FUNCTION_BLOCK SufficientFeedFlow (* CAT Function Block Type *)
  (* Standard: 61499-2 *)
  (* Version 0.0, 9/23/2026, Schneider Electric, template *)
  PACKAGE SE.Nereda;
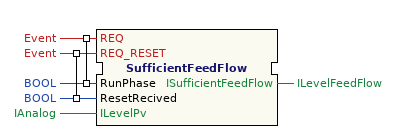
  EVENT_INPUT
    REQ WITH RunPhase; (* Normal Execution Request *)
    REQ_RESET WITH ResetRecived;
  END_EVENT
  VAR_INPUT
    RunPhase : BOOL;
    ResetRecived : BOOL;
  END_VAR
  SOCKETS
    ILevelPv : IAnalog;
  END_SOCKETS
  PLUGS
    ISufficientFeedFlow : ILevelFeedFlow;
  END_PLUGS
  FBS
    SufficientFeedFlow : SufficientFeedFlowBasic;
    E_DELAY : E_DELAY;
    dintToTime : dintToTime;
    IThis : SufficientFeedFlow_HMI(QI := TRUE);
    plcStart1 : plcStart(Prio := 100);
    MUL1 : MUL_112C76C471B7A99C2(IN2 := 1000); {SET_ATTRIBUTE(Configuration.GenericFBType.InterfaceParams, Runtime.Standard#CNT:=2;IN${CNT$}:DINT)}
  END_FBS
  EVENT_CONNECTIONS
    SufficientFeedFlow.CEB292B2283171B2 TO E_DELAY.START;
    SufficientFeedFlow.613F54422BA47101 TO E_DELAY.STOP;
    E_DELAY.EO TO SufficientFeedFlow.9849BF7793E3CBCD;
    REQ TO SufficientFeedFlow.C437AAA8069F1FCB;
    REQ_RESET TO SufficientFeedFlow.B4D22D015D718341;
    dintToTime.CNF TO SufficientFeedFlow.C437AAA8069F1FCB;
    SufficientFeedFlow.AB0236918B6AB7A8 TO ISufficientFeedFlow.CC9428CCDD032224;
    plcStart1.FIRST_INIT TO IThis.2D4FE5DF8F8EB99A;
    plcStart1.REDO_INIT TO IThis.2D4FE5DF8F8EB99A;
    IThis.84013FE241EDAE00 TO SufficientFeedFlow.C437AAA8069F1FCB;
    IThis.2446D9D84A62A6D6 TO plcStart1.ACK_FIRST;
    ILevelPv.REQ TO SufficientFeedFlow.30C32EB006EA4C34;
    IThis.2446D9D84A62A6D6 TO IThis.C95209B68D7D6DBF;
    IThis.84013FE241EDAE00 TO MUL1.REQ;
    MUL1.CNF TO dintToTime.REQ;
  END_CONNECTIONS
  DATA_CONNECTIONS
    RunPhase TO SufficientFeedFlow.90FA4CE95410AC4D;
    ResetRecived TO SufficientFeedFlow.BF5A6785A8565660;
    dintToTime.TimeValue TO SufficientFeedFlow.52D7FB60C38DD9A8;
    SufficientFeedFlow.BE8006DB0CA17265 TO E_DELAY.DT;
    SufficientFeedFlow.F365867250E66A90 TO ISufficientFeedFlow.102CC7A878D73816;
    SufficientFeedFlow.81FE2D2793117977 TO ISufficientFeedFlow.74D3D4DE3ED1D6B7;
    SufficientFeedFlow.60ECB844CED0E64F TO ISufficientFeedFlow.B6B46A0A077DA337;
    SufficientFeedFlow.17DD066F42AD1878 TO ISufficientFeedFlow.957DAAEC5C0D7635;
    IThis.92D95F3FA9CA83CC TO SufficientFeedFlow.9A9AE032169D4A25;
    ILevelPv.Value TO SufficientFeedFlow.BCE3C25201AA8B6A;
    IThis.89CCEFB9E386C33A TO MUL1.IN1;
    MUL1.OUT TO dintToTime.DintTime;
  END_CONNECTIONS
END_FUNCTION_BLOCK
